PROGRAM MAIN
VAR
END_VAR

END_PROGRAM

(* stored: Version 1.1.0.1, ProductVersion 3.1.0.36
   POU MAIN: Id {8387df1b-6459-4265-8430-c8efd58f406a} *)
